
// ===== library: MasterCopy "VFD_Tags" =====

VAR_GLOBAL   // PLC tag table "VFD_Tags"
   "Status_Word" AT %IW76 : Word;   // Drive Status Word
   "Motor_Rpms_In" AT %IW78 : Int;   // Here if you need it. Not in this block
   "Amps_In" AT %IW82 : UInt;   // Amps feedback from drive
   "Fault_Code" AT %IW84 : Word;   // Fault code from drive
   "Control_Word" AT %QW76 : Word;   // Control word to drive
   "Speed_Out_Hz" AT %QW78 : Int;   // Output Speed setpoint to Drive.
   "Run_Fwd" AT %M0.0 : Bool;
   "Run_Rev" AT %M0.1 : Bool;
   "Reset_Fault" AT %M0.2 : Bool;
   "Enable" AT %M0.3 : Bool;
   "Amps_Out" AT %MD0 : Real;
   "Stop" AT %M0.4 : Bool;
   "Line_Volts_In" AT %IW80 : UInt;   // Line voltage reading from drive
   "Speed_Setpoint_Hz" AT %MD4 : Real;   // Set desired speed in Hz `00.0Hz to 60.0Hz`
   "Freq_Fdbk_In" AT %IW86 : Word;   // Frequency feedback from drive
   "E_Stop" AT %M8.0 : Bool;
END_VAR